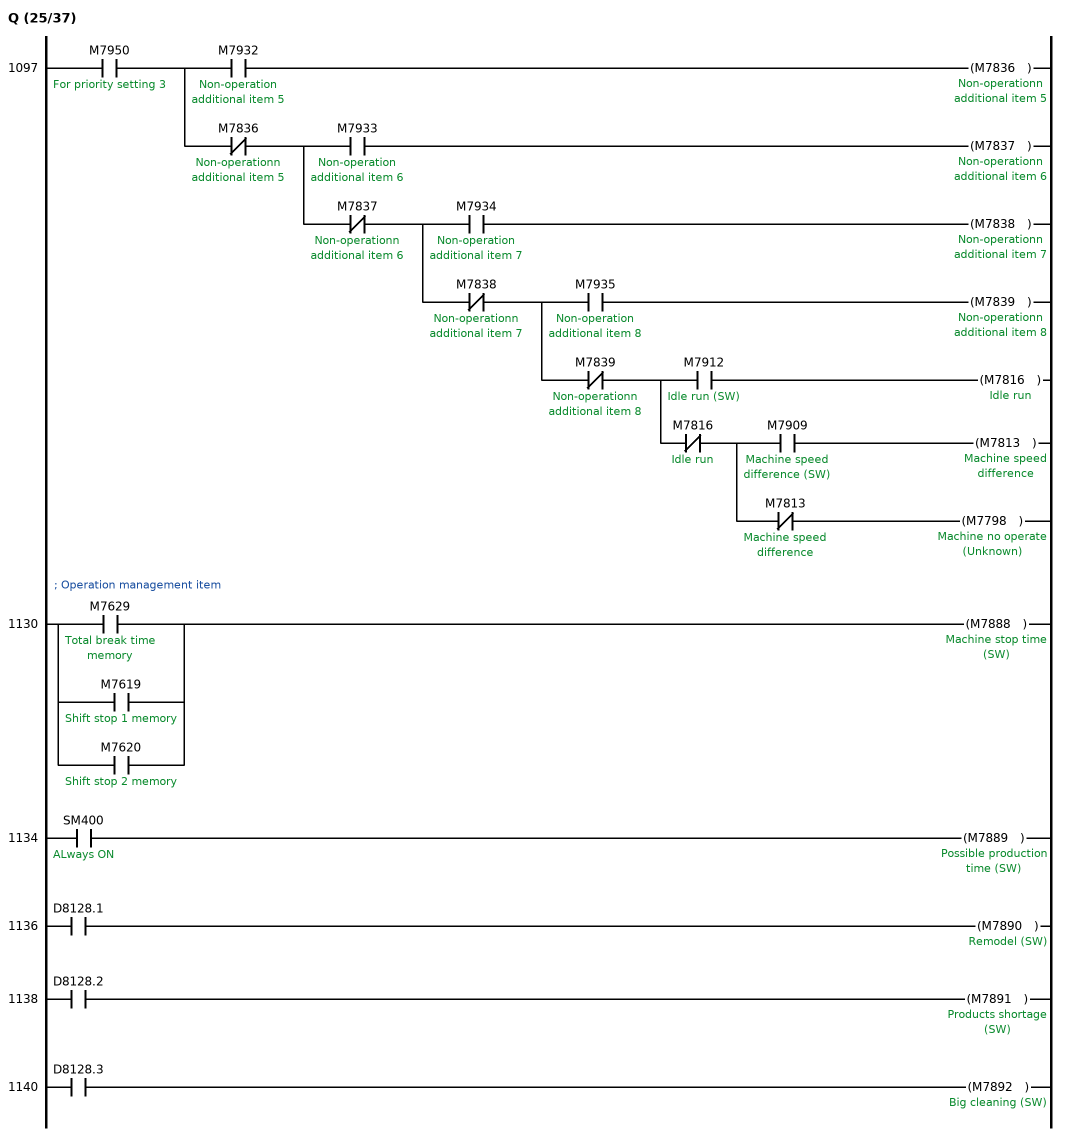
1097  LD      M7950  ; For priority setting 3
      MPS
      AND     M7932  ; Non-operation additional item 5
      OUT     M7836  ; Non-operationn additional item 5
      MPP
      ANI     M7836  ; Non-operationn additional item 5
      MPS
      AND     M7933  ; Non-operation additional item 6
      OUT     M7837  ; Non-operationn additional item 6
      MPP
      ANI     M7837  ; Non-operationn additional item 6
      MPS
      AND     M7934  ; Non-operation additional item 7
      OUT     M7838  ; Non-operationn additional item 7
      MPP
      ANI     M7838  ; Non-operationn additional item 7
      MPS
      AND     M7935  ; Non-operation additional item 8
      OUT     M7839  ; Non-operationn additional item 8
      MPP
      ANI     M7839  ; Non-operationn additional item 8
      MPS
      AND     M7912  ; Idle run (SW)
      OUT     M7816  ; Idle run
      MPP
      ANI     M7816  ; Idle run
      MPS
      AND     M7909  ; Machine speed difference (SW)
      OUT     M7813  ; Machine speed difference
      MPP
      ANI     M7813  ; Machine speed difference
      OUT     M7798  ; Machine no operate (Unknown)
; Operation management item
1130  LD      M7629  ; Total break time memory
      OR      M7619  ; Shift stop 1 memory
      OR      M7620  ; Shift stop 2 memory
      OUT     M7888  ; Machine stop time (SW)
1134  LD      SM400  ; ALways ON
      OUT     M7889  ; Possible production time (SW)
1136  LD      D8128.1
      OUT     M7890  ; Remodel (SW)
1138  LD      D8128.2
      OUT     M7891  ; Products shortage (SW)
1140  LD      D8128.3
      OUT     M7892  ; Big cleaning (SW)
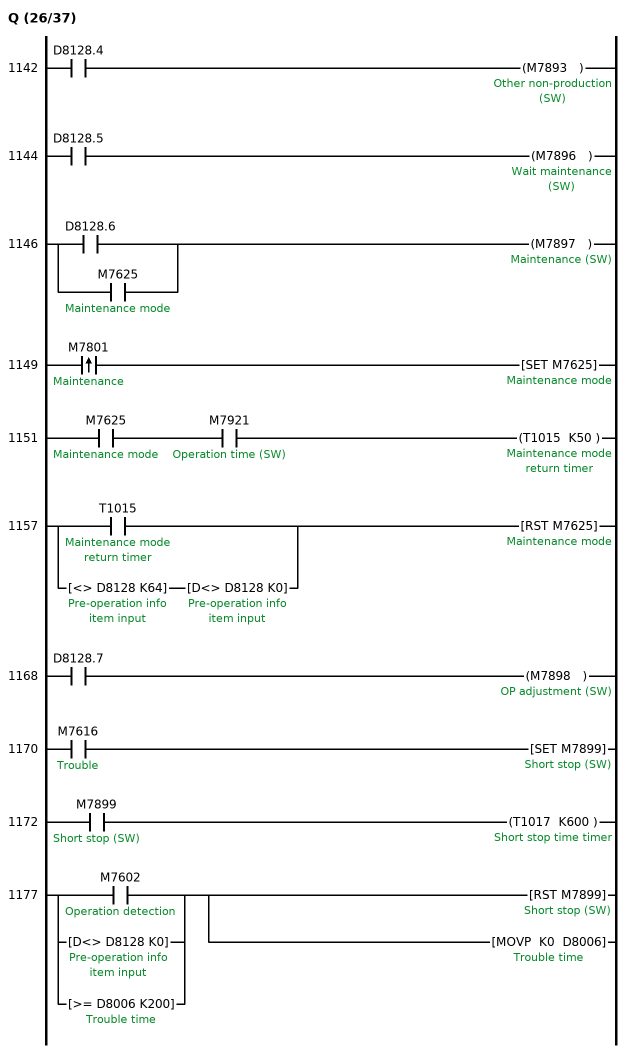
1142  LD      D8128.4
      OUT     M7893  ; Other non-production (SW)
1144  LD      D8128.5
      OUT     M7896  ; Wait maintenance (SW)
1146  LD      D8128.6
      OR      M7625  ; Maintenance mode
      OUT     M7897  ; Maintenance (SW)
1149  LDP     M7801  ; Maintenance
      SET     M7625  ; Maintenance mode
1151  LD      M7625  ; Maintenance mode
      AND     M7921  ; Operation time (SW)
      OUT     T1015 K50  ; Maintenance mode return timer
1157  LD      T1015  ; Maintenance mode return timer
      LD<>    D8128 K64  ; Pre-operation info item input
      ANDD<>  D8128 K0  ; Pre-operation info item input
      ORB
      RST     M7625  ; Maintenance mode
1168  LD      D8128.7
      OUT     M7898  ; OP adjustment (SW)
1170  LD      M7616  ; Trouble
      SET     M7899  ; Short stop (SW)
1172  LD      M7899  ; Short stop (SW)
      OUT     T1017 K600  ; Short stop time timer
1177  LD      M7602  ; Operation detection
      ORD<>   D8128 K0  ; Pre-operation info item input
      OR>=    D8006 K200  ; Trouble time
      RST     M7899  ; Short stop (SW)
      MOVP    K0 D8006
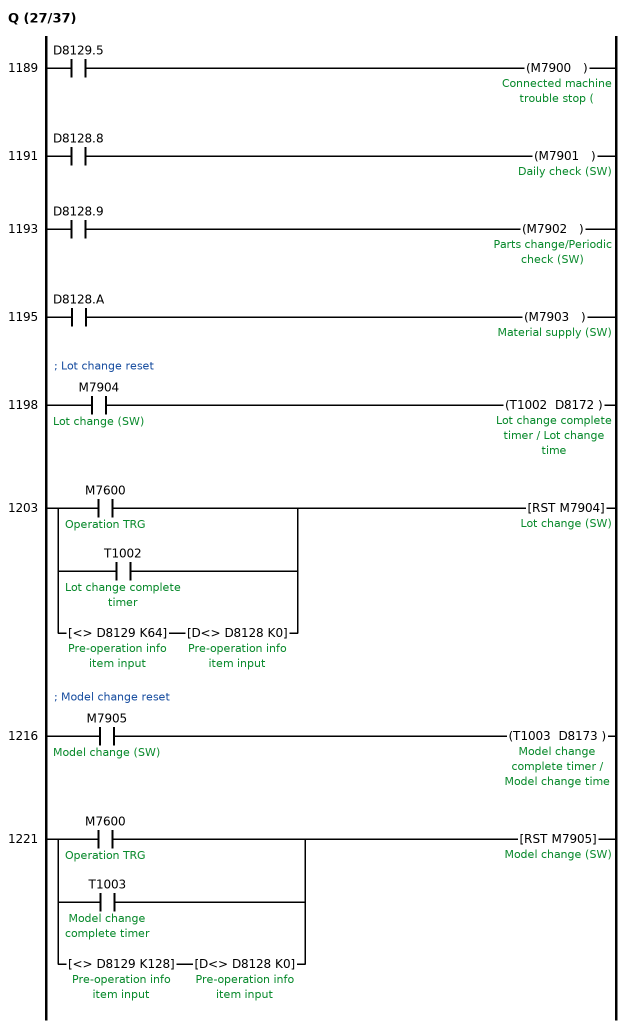
1189  LD      D8129.5
      OUT     M7900  ; Connected machine trouble stop (
1191  LD      D8128.8
      OUT     M7901  ; Daily check (SW)
1193  LD      D8128.9
      OUT     M7902  ; Parts change/Periodic check (SW)
1195  LD      D8128.A
      OUT     M7903  ; Material supply (SW)
; Lot change reset
1198  LD      M7904  ; Lot change (SW)
      OUT     T1002 D8172  ; Lot change complete timer / Lot change time
1203  LD      M7600  ; Operation TRG
      OR      T1002  ; Lot change complete timer
      LD<>    D8129 K64  ; Pre-operation info item input
      ANDD<>  D8128 K0  ; Pre-operation info item input
      ORB
      RST     M7904  ; Lot change (SW)
; Model change reset
1216  LD      M7905  ; Model change (SW)
      OUT     T1003 D8173  ; Model change complete timer / Model change time
1221  LD      M7600  ; Operation TRG
      OR      T1003  ; Model change complete timer
      LD<>    D8129 K128  ; Pre-operation info item input
      ANDD<>  D8128 K0  ; Pre-operation info item input
      ORB
      RST     M7905  ; Model change (SW)
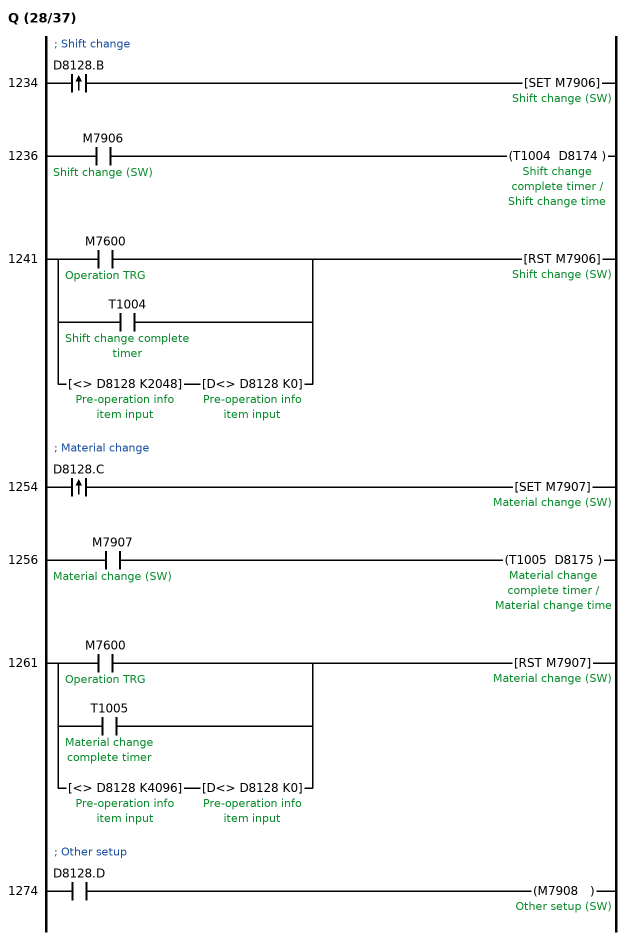
; Shift change
1234  LDP     D8128.B
      SET     M7906  ; Shift change (SW)
1236  LD      M7906  ; Shift change (SW)
      OUT     T1004 D8174  ; Shift change complete timer / Shift change time
1241  LD      M7600  ; Operation TRG
      OR      T1004  ; Shift change complete timer
      LD<>    D8128 K2048  ; Pre-operation info item input
      ANDD<>  D8128 K0  ; Pre-operation info item input
      ORB
      RST     M7906  ; Shift change (SW)
; Material change
1254  LDP     D8128.C
      SET     M7907  ; Material change (SW)
1256  LD      M7907  ; Material change (SW)
      OUT     T1005 D8175  ; Material change complete timer / Material change time
1261  LD      M7600  ; Operation TRG
      OR      T1005  ; Material change complete timer
      LD<>    D8128 K4096  ; Pre-operation info item input
      ANDD<>  D8128 K0  ; Pre-operation info item input
      ORB
      RST     M7907  ; Material change (SW)
; Other setup
1274  LD      D8128.D
      OUT     M7908  ; Other setup (SW)
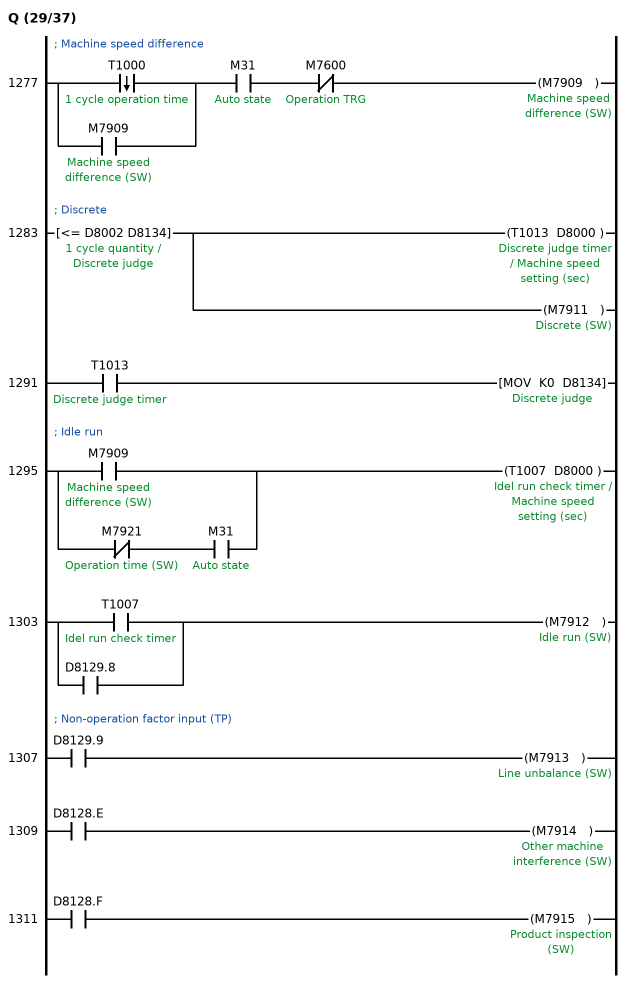
; Machine speed difference
1277  LDF     T1000  ; 1 cycle operation time
      OR      M7909  ; Machine speed difference (SW)
      AND     M31  ; Auto state
      ANI     M7600  ; Operation TRG
      OUT     M7909  ; Machine speed difference (SW)
; Discrete
1283  LD<=    D8002 D8134  ; 1 cycle quantity / Discrete judge
      OUT     T1013 D8000  ; Discrete judge timer / Machine speed setting (sec)
      OUT     M7911  ; Discrete (SW)
1291  LD      T1013  ; Discrete judge timer
      MOV     K0 D8134
; Idle run
1295  LD      M7909  ; Machine speed difference (SW)
      LDI     M7921  ; Operation time (SW)
      AND     M31  ; Auto state
      ORB
      OUT     T1007 D8000  ; Idel run check timer / Machine speed setting (sec)
1303  LD      T1007  ; Idel run check timer
      OR      D8129.8
      OUT     M7912  ; Idle run (SW)
; Non-operation factor input (TP)
1307  LD      D8129.9
      OUT     M7913  ; Line unbalance (SW)
1309  LD      D8128.E
      OUT     M7914  ; Other machine interference (SW)
1311  LD      D8128.F
      OUT     M7915  ; Product inspection (SW)
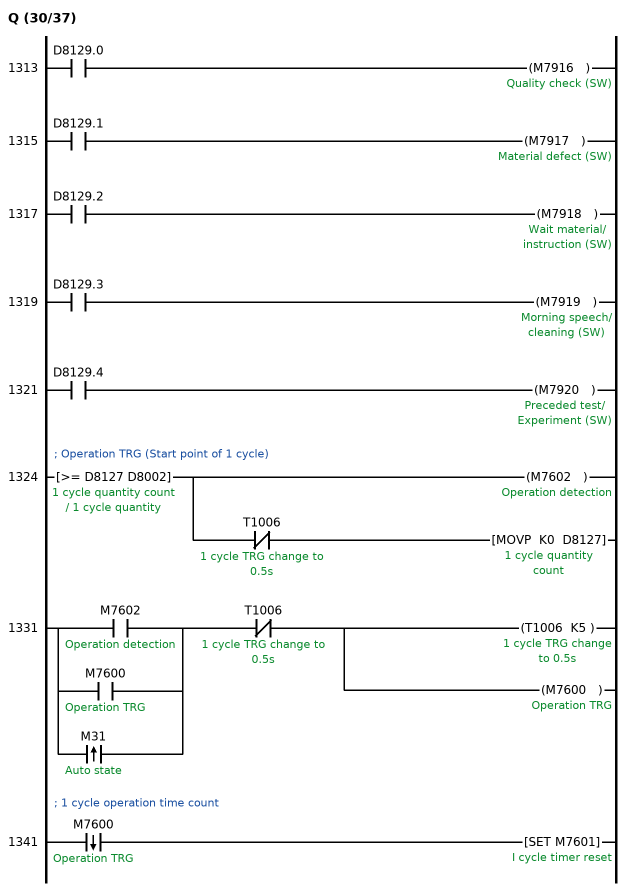
1313  LD      D8129.0
      OUT     M7916  ; Quality check (SW)
1315  LD      D8129.1
      OUT     M7917  ; Material defect (SW)
1317  LD      D8129.2
      OUT     M7918  ; Wait material/instruction (SW)
1319  LD      D8129.3
      OUT     M7919  ; Morning speech/cleaning (SW)
1321  LD      D8129.4
      OUT     M7920  ; Preceded test/Experiment (SW)
; Operation TRG (Start point of 1 cycle)
1324  LD>=    D8127 D8002  ; 1 cycle quantity count / 1 cycle quantity
      OUT     M7602  ; Operation detection
      ANI     T1006  ; 1 cycle TRG change to 0.5s
      MOVP    K0 D8127
1331  LD      M7602  ; Operation detection
      OR      M7600  ; Operation TRG
      ORP     M31  ; Auto state
      ANI     T1006  ; 1 cycle TRG change to 0.5s
      OUT     T1006 K5  ; 1 cycle TRG change to 0.5s
      OUT     M7600  ; Operation TRG
; 1 cycle operation time count
1341  LDF     M7600  ; Operation TRG
      SET     M7601  ; I cycle timer reset
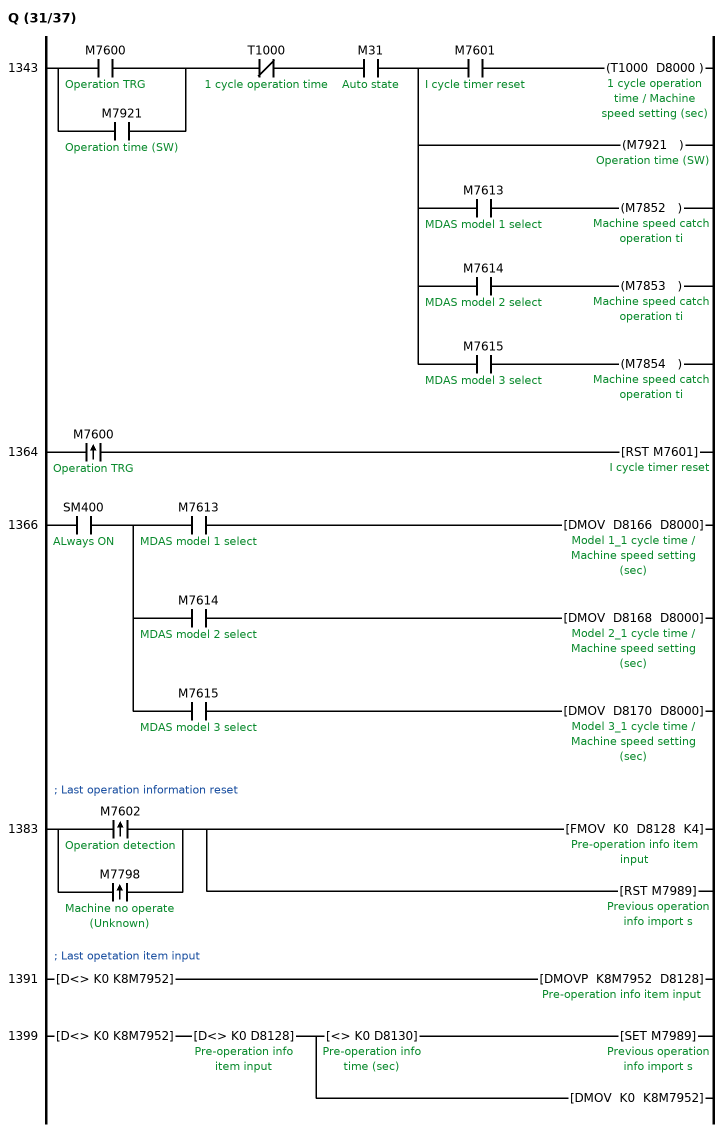
1343  LD      M7600  ; Operation TRG
      OR      M7921  ; Operation time (SW)
      ANI     T1000  ; 1 cycle operation time
      AND     M31  ; Auto state
      MPS
      AND     M7601  ; I cycle timer reset
      OUT     T1000 D8000  ; 1 cycle operation time / Machine speed setting (sec)
      MPP
      OUT     M7921  ; Operation time (SW)
      MPS
      AND     M7613  ; MDAS model 1 select
      OUT     M7852  ; Machine speed catch operation ti
      MRD
      AND     M7614  ; MDAS model 2 select
      OUT     M7853  ; Machine speed catch operation ti
      MPP
      AND     M7615  ; MDAS model 3 select
      OUT     M7854  ; Machine speed catch operation ti
1364  LDP     M7600  ; Operation TRG
      RST     M7601  ; I cycle timer reset
1366  LD      SM400  ; ALways ON
      MPS
      AND     M7613  ; MDAS model 1 select
      DMOV    D8166 D8000
      MRD
      AND     M7614  ; MDAS model 2 select
      DMOV    D8168 D8000
      MPP
      AND     M7615  ; MDAS model 3 select
      DMOV    D8170 D8000
; Last operation information reset
1383  LDP     M7602  ; Operation detection
      ORP     M7798  ; Machine no operate (Unknown)
      FMOV    K0 D8128 K4
      RST     M7989  ; Previous operation info import s
; Last opetation item input
1391  LDD<>   K0 K8M7952  ; TP (Lunch break, Shift stop)
      DMOVP   K8M7952 D8128
1399  LDD<>   K0 K8M7952  ; TP (Lunch break, Shift stop)
      ANDD<>  K0 D8128  ; Pre-operation info item input
      MPS
      AND<>   K0 D8130  ; Pre-operation info time (sec)
      SET     M7989  ; Previous operation info import s
      MPP
      DMOV    K0 K8M7952
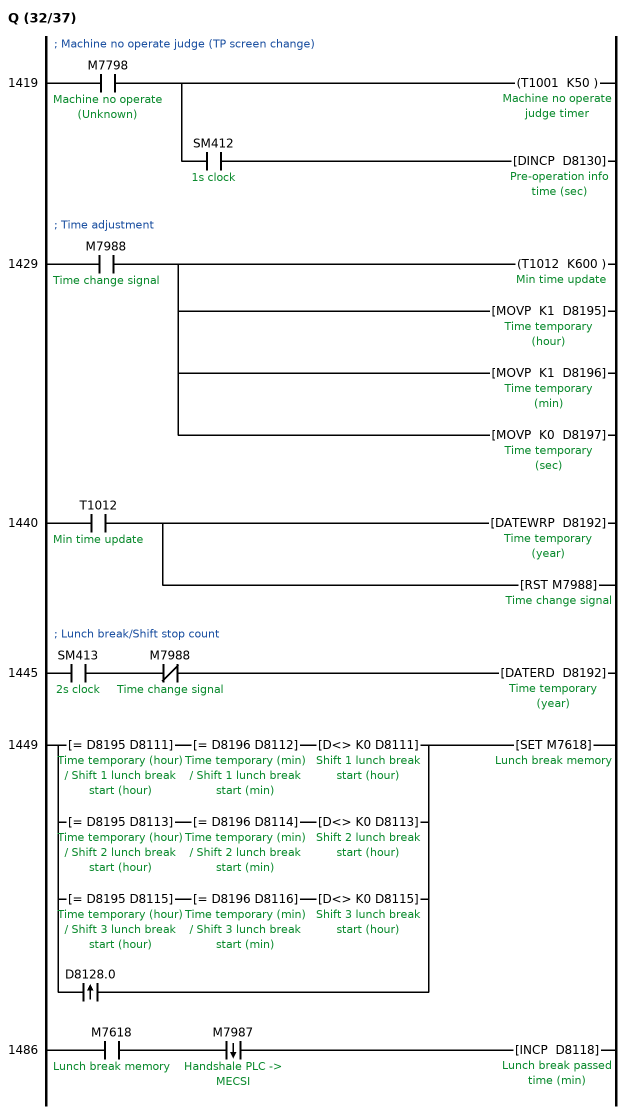
; Machine no operate judge (TP screen change)
1419  LD      M7798  ; Machine no operate (Unknown)
      OUT     T1001 K50  ; Machine no operate judge timer
      AND     SM412  ; 1s clock
      DINCP   D8130
; Time adjustment
1429  LD      M7988  ; Time change signal
      OUT     T1012 K600  ; Min time update
      MOVP    K1 D8195  ; Time temporary (hour)
      MOVP    K1 D8196  ; Time temporary (min)
      MOVP    K0 D8197  ; Time temporary (sec)
1440  LD      T1012  ; Min time update
      DATEWRP D8192  ; Time temporary (year)
      RST     M7988  ; Time change signal
; Lunch break/Shift stop count
1445  LD      SM413  ; 2s clock
      ANI     M7988  ; Time change signal
      DATERD  D8192
1449  LD=     D8195 D8111  ; Time temporary (hour) / Shift 1 lunch break start (hour)
      AND=    D8196 D8112  ; Time temporary (min) / Shift 1 lunch break start (min)
      ANDD<>  K0 D8111  ; Shift 1 lunch break start (hour)
      LD=     D8195 D8113  ; Time temporary (hour) / Shift 2 lunch break start (hour)
      AND=    D8196 D8114  ; Time temporary (min) / Shift 2 lunch break start (min)
      ANDD<>  K0 D8113  ; Shift 2 lunch break start (hour)
      ORB
      LD=     D8195 D8115  ; Time temporary (hour) / Shift 3 lunch break start (hour)
      AND=    D8196 D8116  ; Time temporary (min) / Shift 3 lunch break start (min)
      ANDD<>  K0 D8115  ; Shift 3 lunch break start (hour)
      ORB
      ORP     D8128.0
      SET     M7618  ; Lunch break memory
1486  LD      M7618  ; Lunch break memory
      ANDF    M7987  ; Handshale PLC -> MECSI
      INCP    D8118  ; Lunch break passed time (min)
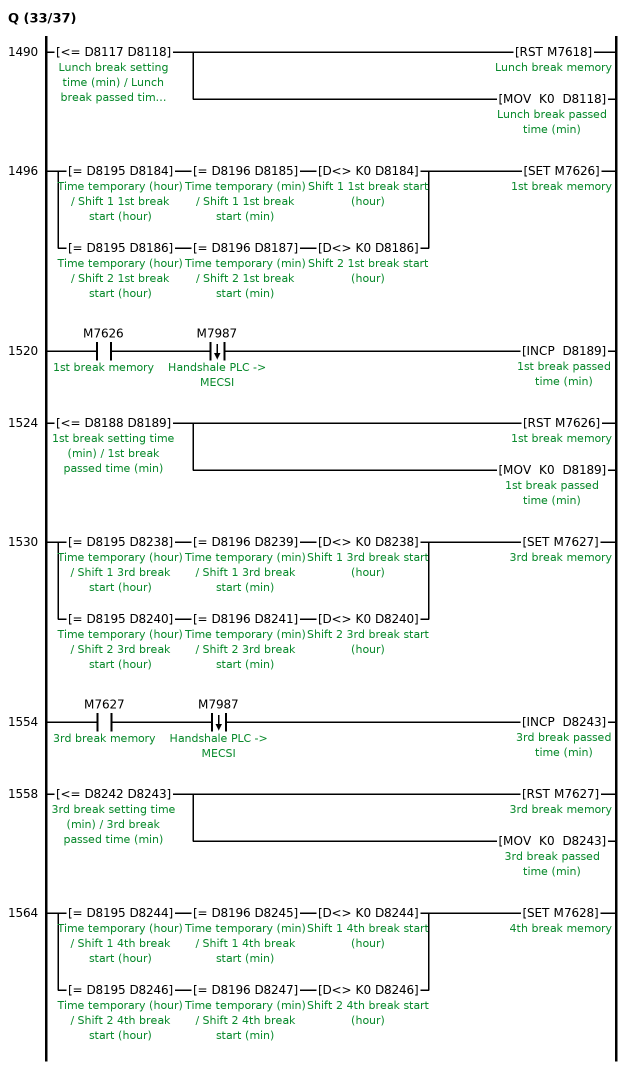
1490  LD<=    D8117 D8118  ; Lunch break setting time (min) / Lunch break passed time (min)
      RST     M7618  ; Lunch break memory
      MOV     K0 D8118
1496  LD=     D8195 D8184  ; Time temporary (hour) / Shift 1 1st break start (hour)
      AND=    D8196 D8185  ; Time temporary (min) / Shift 1 1st break start (min)
      ANDD<>  K0 D8184  ; Shift 1 1st break start (hour)
      LD=     D8195 D8186  ; Time temporary (hour) / Shift 2 1st break start (hour)
      AND=    D8196 D8187  ; Time temporary (min) / Shift 2 1st break start (min)
      ANDD<>  K0 D8186  ; Shift 2 1st break start (hour)
      ORB
      SET     M7626  ; 1st break memory
1520  LD      M7626  ; 1st break memory
      ANDF    M7987  ; Handshale PLC -> MECSI
      INCP    D8189  ; 1st break passed time (min)
1524  LD<=    D8188 D8189  ; 1st break setting time (min) / 1st break passed time (min)
      RST     M7626  ; 1st break memory
      MOV     K0 D8189
1530  LD=     D8195 D8238  ; Time temporary (hour) / Shift 1 3rd break start (hour)
      AND=    D8196 D8239  ; Time temporary (min) / Shift 1 3rd break start (min)
      ANDD<>  K0 D8238  ; Shift 1 3rd break start (hour)
      LD=     D8195 D8240  ; Time temporary (hour) / Shift 2 3rd break start (hour)
      AND=    D8196 D8241  ; Time temporary (min) / Shift 2 3rd break start (min)
      ANDD<>  K0 D8240  ; Shift 2 3rd break start (hour)
      ORB
      SET     M7627  ; 3rd break memory
1554  LD      M7627  ; 3rd break memory
      ANDF    M7987  ; Handshale PLC -> MECSI
      INCP    D8243  ; 3rd break passed time (min)
1558  LD<=    D8242 D8243  ; 3rd break setting time (min) / 3rd break passed time (min)
      RST     M7627  ; 3rd break memory
      MOV     K0 D8243
1564  LD=     D8195 D8244  ; Time temporary (hour) / Shift 1 4th break start (hour)
      AND=    D8196 D8245  ; Time temporary (min) / Shift 1 4th break start (min)
      ANDD<>  K0 D8244  ; Shift 1 4th break start (hour)
      LD=     D8195 D8246  ; Time temporary (hour) / Shift 2 4th break start (hour)
      AND=    D8196 D8247  ; Time temporary (min) / Shift 2 4th break start (min)
      ANDD<>  K0 D8246  ; Shift 2 4th break start (hour)
      ORB
      SET     M7628  ; 4th break memory
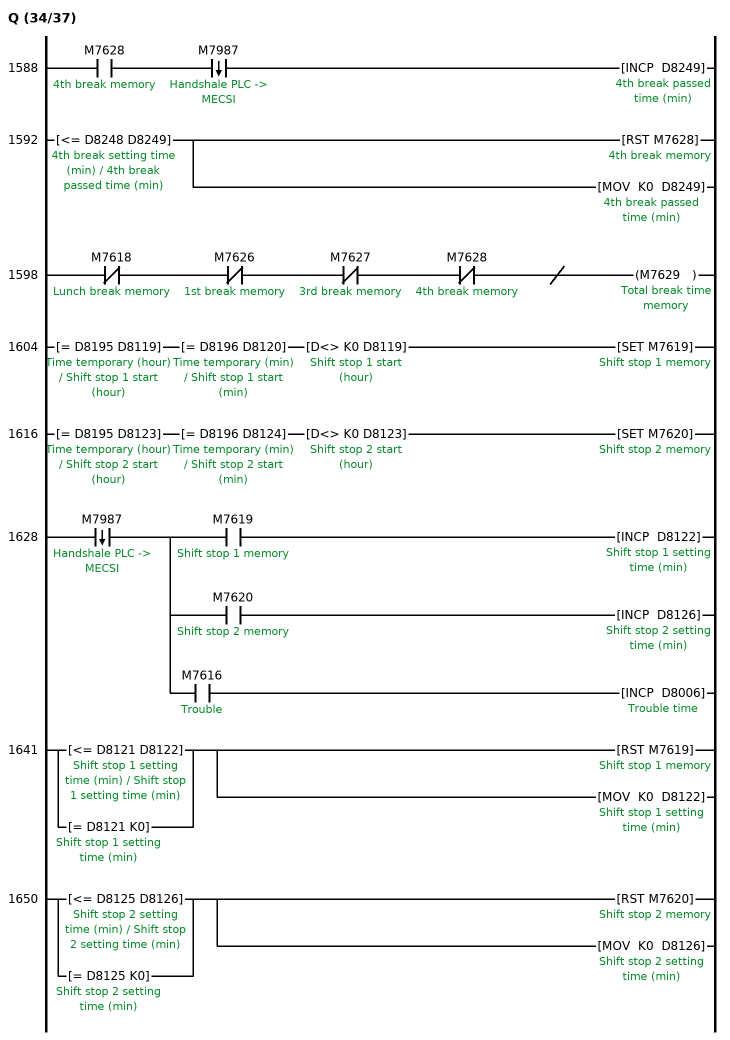
1588  LD      M7628  ; 4th break memory
      ANDF    M7987  ; Handshale PLC -> MECSI
      INCP    D8249  ; 4th break passed time (min)
1592  LD<=    D8248 D8249  ; 4th break setting time (min) / 4th break passed time (min)
      RST     M7628  ; 4th break memory
      MOV     K0 D8249
1598  LDI     M7618  ; Lunch break memory
      ANI     M7626  ; 1st break memory
      ANI     M7627  ; 3rd break memory
      ANI     M7628  ; 4th break memory
      INV
      OUT     M7629  ; Total break time memory
1604  LD=     D8195 D8119  ; Time temporary (hour) / Shift stop 1 start (hour)
      AND=    D8196 D8120  ; Time temporary (min) / Shift stop 1 start (min)
      ANDD<>  K0 D8119  ; Shift stop 1 start (hour)
      SET     M7619  ; Shift stop 1 memory
1616  LD=     D8195 D8123  ; Time temporary (hour) / Shift stop 2 start (hour)
      AND=    D8196 D8124  ; Time temporary (min) / Shift stop 2 start (min)
      ANDD<>  K0 D8123  ; Shift stop 2 start (hour)
      SET     M7620  ; Shift stop 2 memory
1628  LDF     M7987  ; Handshale PLC -> MECSI
      MPS
      AND     M7619  ; Shift stop 1 memory
      INCP    D8122  ; Shift stop 1 setting time (min)
      MRD
      AND     M7620  ; Shift stop 2 memory
      INCP    D8126  ; Shift stop 2 setting time (min)
      MPP
      AND     M7616  ; Trouble
      INCP    D8006
1641  LD<=    D8121 D8122  ; Shift stop 1 setting time (min) / Shift stop 1 setting time (min)
      OR=     D8121 K0  ; Shift stop 1 setting time (min)
      RST     M7619  ; Shift stop 1 memory
      MOV     K0 D8122
1650  LD<=    D8125 D8126  ; Shift stop 2 setting time (min) / Shift stop 2 setting time (min)
      OR=     D8125 K0  ; Shift stop 2 setting time (min)
      RST     M7620  ; Shift stop 2 memory
      MOV     K0 D8126
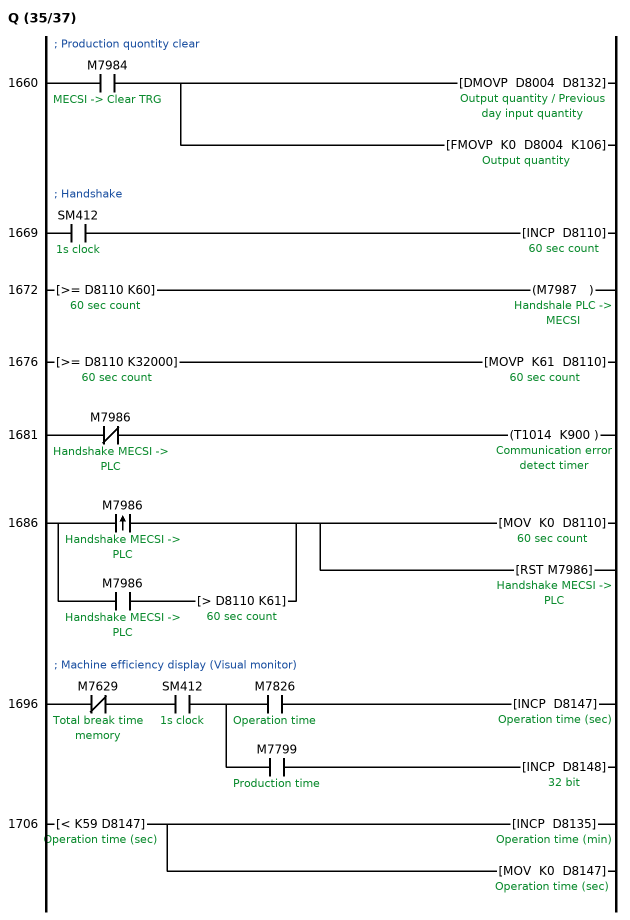
; Production quontity clear
1660  LD      M7984  ; MECSI -> Clear TRG
      DMOVP   D8004 D8132  ; Previous day input quantity
      FMOVP   K0 D8004 K106
; Handshake
1669  LD      SM412  ; 1s clock
      INCP    D8110  ; 60 sec count
1672  LD>=    D8110 K60  ; 60 sec count
      OUT     M7987  ; Handshale PLC -> MECSI
1676  LD>=    D8110 K32000  ; 60 sec count
      MOVP    K61 D8110
1681  LDI     M7986  ; Handshake MECSI -> PLC
      OUT     T1014 K900  ; Communication error detect timer
1686  LDP     M7986  ; Handshake MECSI -> PLC
      LD      M7986  ; Handshake MECSI -> PLC
      AND>    D8110 K61  ; 60 sec count
      ORB
      MOV     K0 D8110
      RST     M7986  ; Handshake MECSI -> PLC
; Machine efficiency display (Visual monitor)
1696  LDI     M7629  ; Total break time memory
      AND     SM412  ; 1s clock
      MPS
      AND     M7826  ; Operation time
      INCP    D8147  ; Operation time (sec)
      MPP
      AND     M7799  ; Production time
      INCP    D8148  ; 32 bit
1706  LD<     K59 D8147  ; Operation time (sec)
      INCP    D8135  ; Operation time (min)
      MOV     K0 D8147
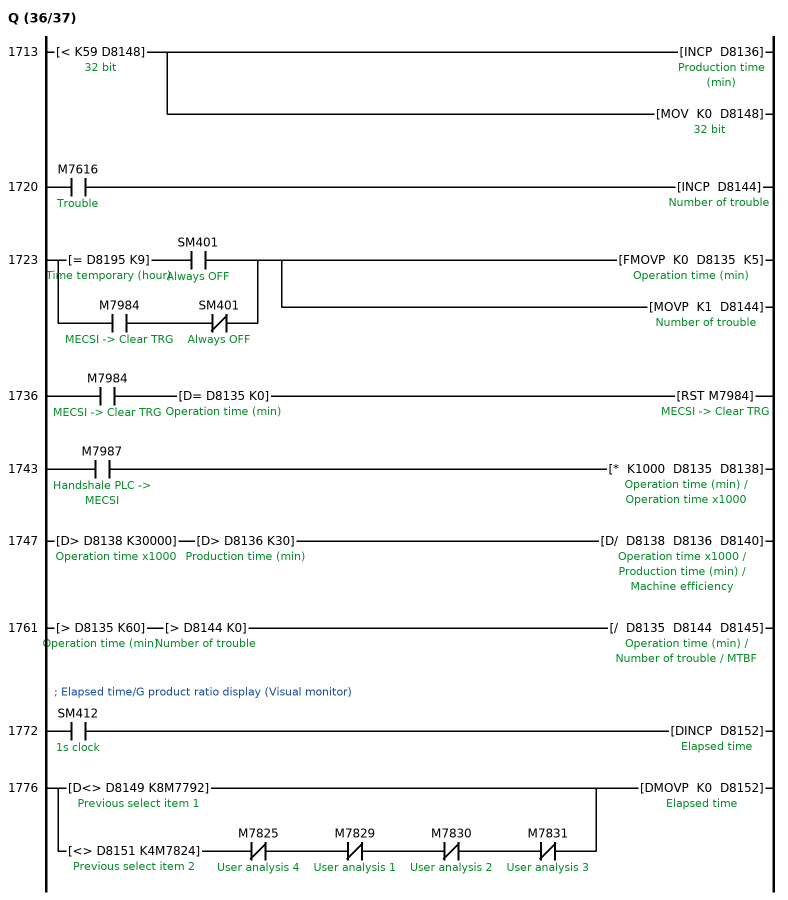
1713  LD<     K59 D8148  ; 32 bit
      INCP    D8136  ; Production time (min)
      MOV     K0 D8148
1720  LD      M7616  ; Trouble
      INCP    D8144  ; Number of trouble
1723  LD=     D8195 K9  ; Time temporary (hour)
      AND     SM401  ; Always OFF
      LD      M7984  ; MECSI -> Clear TRG
      ANI     SM401  ; Always OFF
      ORB
      FMOVP   K0 D8135 K5
      MOVP    K1 D8144
1736  LD      M7984  ; MECSI -> Clear TRG
      ANDD=   D8135 K0  ; Operation time (min)
      RST     M7984  ; MECSI -> Clear TRG
1743  LD      M7987  ; Handshale PLC -> MECSI
      *       K1000 D8135 D8138  ; Operation time x1000
1747  LDD>    D8138 K30000  ; Operation time x1000
      ANDD>   D8136 K30  ; Production time (min)
      D/      D8138 D8136 D8140  ; Machine efficiency
1761  LD>     D8135 K60  ; Operation time (min)
      AND>    D8144 K0  ; Number of trouble
      /       D8135 D8144 D8145  ; MTBF
; Elapsed time/G product ratio display (Visual monitor)
1772  LD      SM412  ; 1s clock
      DINCP   D8152  ; Elapsed time
1776  LDD<>   D8149 K8M7792  ; Previous select item 1 / Machine stop time
      LD<>    D8151 K4M7824  ; Previous select item 2 / Preceded test/Experiment
      ANI     M7825  ; User analysis 4
      ANI     M7829  ; User analysis 1
      ANI     M7830  ; User analysis 2
      ANI     M7831  ; User analysis 3
      ORB
      DMOVP   K0 D8152
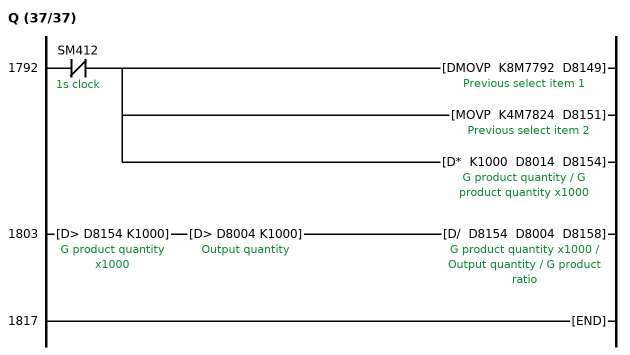
1792  LDI     SM412  ; 1s clock
      DMOVP   K8M7792 D8149
      MOVP    K4M7824 D8151
      D*      K1000 D8014 D8154  ; G product quantity x1000
1803  LDD>    D8154 K1000  ; G product quantity x1000
      ANDD>   D8004 K1000  ; Output quantity
      D/      D8154 D8004 D8158  ; G product ratio
1817  END
END_PROGRAM

// device comments not shown above
M7603  ; Auto check PLS
M7604  ; Input quantity clear FLG
M7605  ; Handshake PLF
M7607  ; Delay check PLF
M7608  ; Operation TRG PLS
M7609  ; Operation TRG PLF
M7611  ; Auto stop check wait PLS
M7617  ; Operation detection PLF
M7622  ; Machine no operate PLS
M7783  ; Alarm call 1
M7784  ; Alarm call 2
M7785  ; Alarm call 3
M7786  ; Alarm call 4
M7787  ; Alarm call 5
M7788  ; Alarm call 6
M7789  ; Alarm call 7
M7790  ; Alarm call 8
M7791  ; Alarm call 9
M7855  ; Operation detail item 1
M7856  ; Operation detail item 2
M7857  ; Operation detail item 3
M7858  ; Operation detail item 4
M7859  ; Operation detail item 5
M7860  ; Operation detail item 6
M7861  ; Operation detail item 7
M7862  ; Operation detail item 8
M7863  ; Operation detail item 9
M7864  ; Operation detail item 10
M7865  ; Off-line setup detail 1
M7866  ; Off-line setup detail 2
M7867  ; Off-line setup detail 3
M7868  ; Off-line setup detail 4
M7869  ; Off-line setup detail 5
M7870  ; Off-line setup detail 6
M7871  ; Off-line setup detail 7
M7872  ; Maintenance (No priority)
M7873  ; OP adjustment (No priority)
M7874  ; Daily check (No priority)
M7875  ; Material supply (No priority)
M7876  ; Lot change (No priority)
M7877  ; Model change (No priority)
M7878  ; Shift change (No priority)
M7879  ; Material change (No priority)
M7880  ; Other setup (No priority)
M7894  ; Use reserve (SW)
M7895  ; Use reserve (SW)
M7936  ; Operation detail SW 1
M7937  ; Operation detail SW 2
M7938  ; Operation detail SW 3
M7939  ; Operation detail SW 4
M7940  ; Operation detail SW 5
M7941  ; Operation detail SW 6
M7942  ; Operation detail SW 7
M7943  ; Operation detail SW 8
M7944  ; Operation detail SW 9
M7945  ; Operation detail SW 10
M7951  ; For priority setting 4
M7953  ; TP (Remode)
M7954  ; TP (Products shortage)
M7955  ; TP (Big cleaning)
M7956  ; TP (Other non-production
M7957  ; TP (Wait maintenance)
M7958  ; TP (Maintenance)
M7959  ; TP (Adjustment)
M7960  ; TP (Daily check)
M7961  ; TP (Periodic maintenance)
M7962  ; TP (Material supply)
M7963  ; TP (Shift change)
M7964  ; TP (Material change)
M7965  ; TP (Other setup)
M7966  ; TP (Machine interference)
M7967  ; TP (Product inspection)
M7968  ; TP (Quality check)
M7969  ; TP (Material defect)
M7970  ; TP (Wait material/Instruction)
M7971  ; TP (Morning speech)
M7972  ; TP (Preceded test/Experiment)
M7973  ; TP (Machine interference stop)
M7974  ; TP (Lot change)
M7975  ; TP (Model change)
M7976  ; TP (Idel run)
M7977  ; TP (Line unbalance)
M7978  ; TP (Non-production item 1)
M7979  ; TP (Non-production item 2)
M7980  ; TP (Non-operation item 1)
M7981  ; TP (Non-operation item 2)
M7982  ; TP (Non-operation item 3)
M7983  ; TP (Non-operation item 4)
P20  ; 下ﾘｰﾄﾞｼﾌﾄ
P22  ; 下ﾘｰﾄﾞst8ｼﾌﾄ
P26  ; 上ﾘｰﾄﾞｼﾌﾄ
P30  ; ﾃｰﾌﾞﾙ上ｼﾌﾄ
P52  ; 原点ﾓﾆﾀ
P54  ; 表示中ｽｸﾘｰﾝ･ｶﾚﾝﾀﾞ書込み
P55  ; ﾃﾞｰﾀｸﾘｱ
P56  ; ﾃﾞｰﾀ書き換え許可
P60  ; 補助ﾓｰﾄﾞ設定
P62  ; ﾃﾞﾊﾞｲｽﾓﾆﾀ
P64  ; 稼動ﾃﾞｰﾀ
P66  ; ｶｳﾝﾀ
P70  ; 品種選択
P72  ; 品種情報設定
P90  ; 品種Aﾊﾟﾚｯﾄ演算
P91  ; 品種Bﾊﾟﾚｯﾄ演算
